FUNCTION_BLOCK FB_ProBoxElement2MotorEmulation EXTENDS FB_ElementConvEmulation
(**************************************************************************************
 * 	Application		:	BoxControl Framework
 *	Revision		:	$Revision:  $
 *	Revision date	:	$Date: $
 *	Last changed by	:	$Author: $
 *	URL				:	$URL: $
 *
 *	Purpose			:	Emulation of probox two motor element.
 *
 * ------------------------------------------------------------------------------------
 *	Copyright Swisslog [IP AG], Switzerland. All rights reserved.
 * 
 * ------------------------------------------------------------------------------------
 *	
 * 	Revision History: 
 *
 * 	VERSION			DATE			INITIALS			DESCRIPTION
 *
 **************************************************************************************)
VAR
	pElement						: POINTER TO FB_ProBoxElement2Motor; // Address to element
	rElement						: REFERENCE TO FB_ProBoxElement2Motor; // Reference to element	
END_VAR

(**************************************************************************************************************
   Initialization
***************************************************************************************************************)
A_Init();

(**************************************************************************************************************
   Update reference
***************************************************************************************************************)
A_UpdateReference();

(**************************************************************************************************************
   Emulation
***************************************************************************************************************)
// If emulation element is initialized
IF ElementData.Init THEN
	
	// Update real data
	M_UpdateRealObjectData();	
	
	//Set emulation speed	
	rElement.P_EmuSpeed	:= ProBoxSystem.EMULATION_SPEED;
	
	// Overwrite inputs
	A_OverWriteInputs();

END_IF

ACTION A_Init:
(**************************************************************************************
 * 	NAME		A_Init
 * 	FUNCTION	Initialize emulated dummy element
 **************************************************************************************)

// If element is not initialized
IF NOT ElementData.Init THEN

	// Check that linked element number is valid
	IF eElementNumber > E_ElementNumber.E_BEGIN_ELEMENT AND
	   eElementNumber < E_ElementNumber.E_END_ELEMENT THEN
		
			// Check that the real module is initialized
			IF F_IsElementInitialized(eElementNumber) THEN
				// Module is initialized
				ElementData.Init := TRUE;
				
				// Send debug message
				DebugMsg := CONCAT('Initialization done. Element: ', ElementRegistry[eElementNumber].ElementName);
				fbDebugMsg.M_SendInfoMsg(DebugMsg);
				
				// Initialize real module
				F_InitializeElement(eElementNumber := eElementNumber);
			END_IF
	END_IF
END_IF
END_ACTION

ACTION A_OverWriteInputs:
(**************************************************************************************
* 	NAME		A_OverWriteInputs
* 	FUNCTION	Overwrite hardware inputs for emulation
**************************************************************************************)

rElement.HW_Inputs.MotorUnitOK := TRUE;
END_ACTION

ACTION A_UpdateReference:
(**************************************************************************************
 * 	NAME		A_UpdateReference
 * 	FUNCTION	Update reference to real object
 **************************************************************************************)

// Check valid element number
IF eElementNumber > E_ElementNumber.E_BEGIN_ELEMENT AND
   eElementNumber < E_ElementNumber.E_END_ELEMENT THEN

	// Is reference valid  
	IF __ISVALIDREF(ElementRegistry[eElementNumber].rElement) THEN
		// Build address to reference
		pElement := ADR(ElementRegistry[eElementNumber].rElement);

		// If address is possible
		IF pElement <> 0 THEN
			// Build reference to memory
			rElement REF= pElement^;
		ELSE
			// Reinitialize module
			ElementData.Init := FALSE;
		END_IF
	ELSE
		// Reinitialize module
		ElementData.Init := FALSE;
	END_IF
END_IF
END_ACTION

END_FUNCTION_BLOCK

(* stored: Version 1.1.0.1, ProductVersion 3.1.4024.9
   POU FB_ProBoxElement2MotorEmulation: Id {abdc8ccc-c4e8-4e11-9ac3-817670386e0a}, SpecialFunc None
   Action A_Init: Id {5f5349f0-9689-4f43-a097-6842aaaa6262}
   Action A_OverWriteInputs: Id {28f7f3fb-ffc6-40ff-ae14-7e9e6e4ba3a2}
   Action A_UpdateReference: Id {0940c9e0-09b9-45ce-a4a5-ec89fcac8d33} *)
